// TIA Portal V17 export
// export: Created 2023-04-04T13:27:33.4464749Z, ExportSetting WithDefaults, DisplayName Totally Integrated Automation Portal, DisplayVersion V17, DisplayName TIA Portal Openness, DisplayVersion V17, DisplayName TIA Portal Version Control Interface, DisplayVersion V17, DisplayName STEP 7 Professional, DisplayVersion V17, DisplayName STEP 7 Safety, DisplayVersion V17, DisplayName WinCC Advanced, DisplayVersion V17
TYPE "typ_Order_Workpiece_Buttons"
// stored: IsFailsafeCompliant false
   STRUCT
      ldt_ts : LDT;
      s_type : String;
      Workpiece_Parameters : "typ_Workpiece_Parameters";
   END_STRUCT;
   // Workpiece_Parameters.DoOven := true;
   // Workpiece_Parameters.OvenTime := T#4S;
   // Workpiece_Parameters.DoSaw := true;
   // Workpiece_Parameters.SawTime := T#4S;
END_TYPE
